# EPICS autosave request: iocBoot/ioc2/dbSave/23i_BP_Mo_.req
%
% BURT Request File
%
% 23i:BP:Mo:  BPM @ monochromator position
%

file $(DIR)/assy.req ASSY=23i:BP:Mo
file $(DIR)/mtr1.req MTR1=23i:BP:mmo
file $(DIR)/drv1.req DRV1=23i:BP:MOZ
